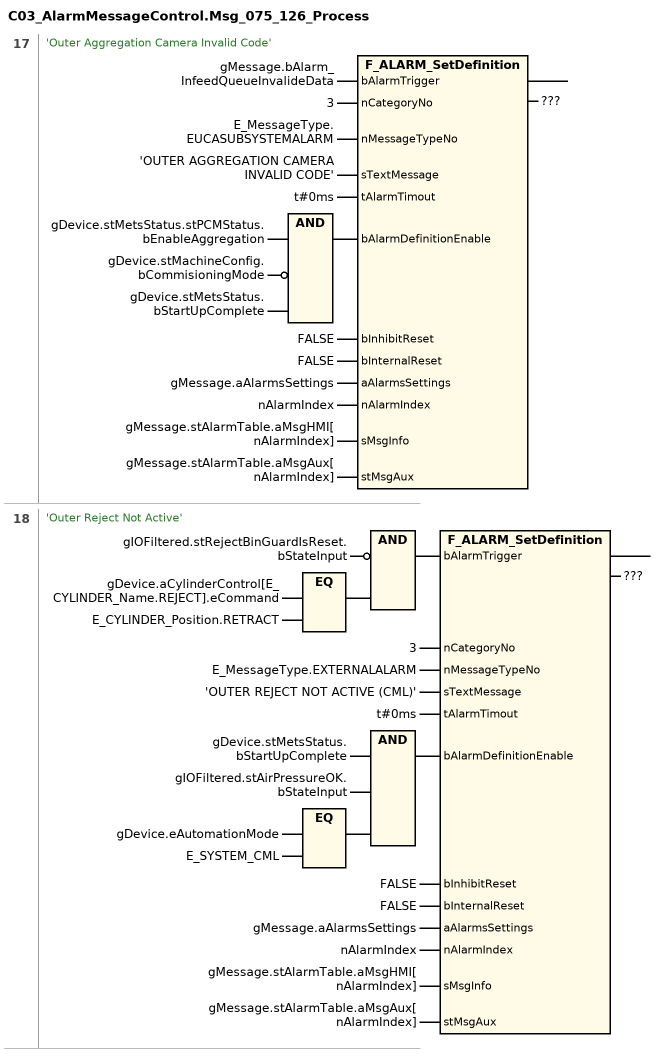
// NETWORK 17
// 'Outer Aggregation Camera Invalid Code'
F_ALARM_SetDefinition(bAlarmTrigger := gMessage.bAlarm_InfeedQueueInvalideData, nCategoryNo := 3, nMessageTypeNo := E_MessageType.EUCASUBSYSTEMALARM, sTextMessage := 'OUTER AGGREGATION CAMERA INVALID CODE', tAlarmTimout := t#0ms, bAlarmDefinitionEnable := gDevice.stMetsStatus.stPCMStatus.bEnableAggregation AND NOT gDevice.stMachineConfig.bCommisioningMode AND gDevice.stMetsStatus.bStartUpComplete, bInhibitReset := FALSE, bInternalReset := FALSE, aAlarmsSettings := gMessage.aAlarmsSettings, nAlarmIndex := nAlarmIndex, sMsgInfo := gMessage.stAlarmTable.aMsgHMI[nAlarmIndex], stMsgAux := gMessage.stAlarmTable.aMsgAux[nAlarmIndex]);

// NETWORK 18
// 'Outer Reject Not Active'
F_ALARM_SetDefinition(bAlarmTrigger := NOT gIOFiltered.stRejectBinGuardIsReset.bStateInput AND gDevice.aCylinderControl[E_CYLINDER_Name.REJECT].eCommand = E_CYLINDER_Position.RETRACT, nCategoryNo := 3, nMessageTypeNo := E_MessageType.EXTERNALALARM, sTextMessage := 'OUTER REJECT NOT ACTIVE (CML)', tAlarmTimout := t#0ms, bAlarmDefinitionEnable := gDevice.stMetsStatus.bStartUpComplete AND gIOFiltered.stAirPressureOK.bStateInput AND gDevice.eAutomationMode = E_SYSTEM_CML, bInhibitReset := FALSE, bInternalReset := FALSE, aAlarmsSettings := gMessage.aAlarmsSettings, nAlarmIndex := nAlarmIndex, sMsgInfo := gMessage.stAlarmTable.aMsgHMI[nAlarmIndex], stMsgAux := gMessage.stAlarmTable.aMsgAux[nAlarmIndex]);

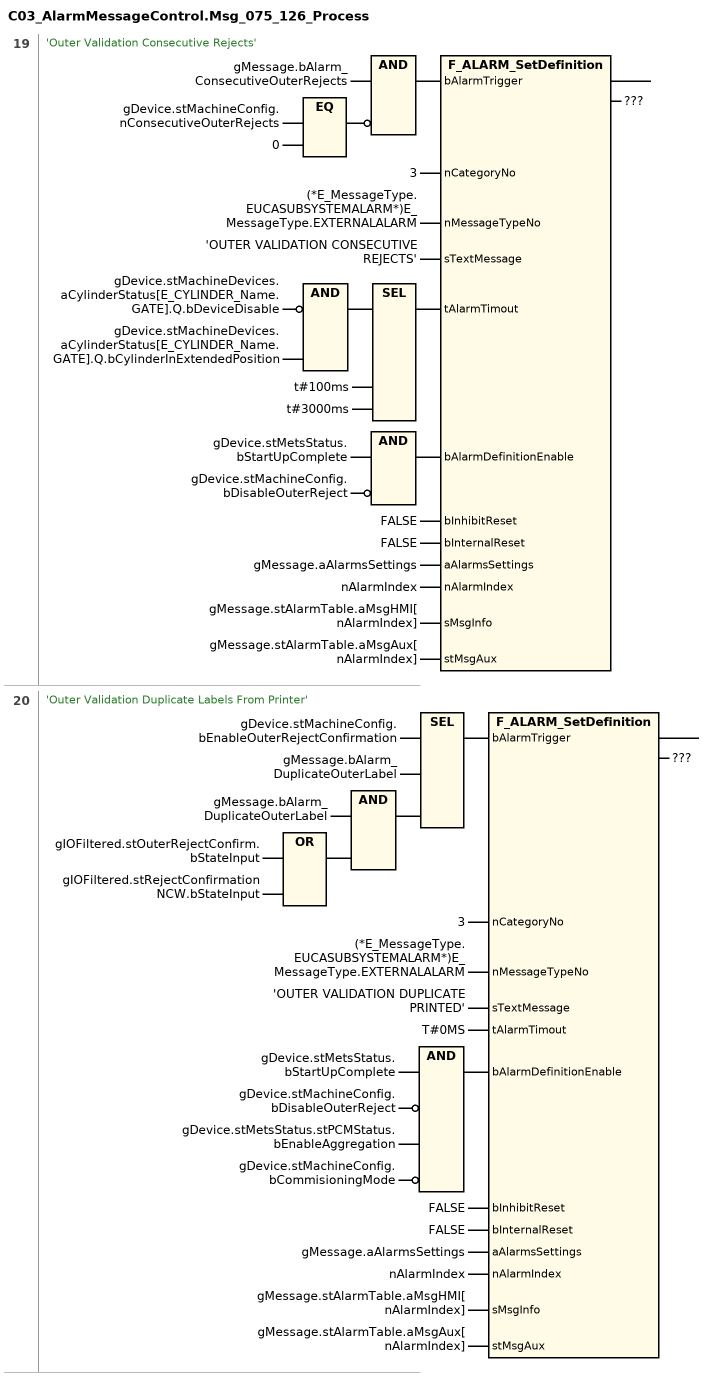
// NETWORK 19
// 'Outer Validation Consecutive Rejects'
F_ALARM_SetDefinition(bAlarmTrigger := gMessage.bAlarm_ConsecutiveOuterRejects AND NOT (gDevice.stMachineConfig.nConsecutiveOuterRejects = 0), nCategoryNo := 3, nMessageTypeNo := (*E_MessageType.EUCASUBSYSTEMALARM*)E_MessageType.EXTERNALALARM, sTextMessage := 'OUTER VALIDATION CONSECUTIVE REJECTS', tAlarmTimout := SEL(NOT gDevice.stMachineDevices.aCylinderStatus[E_CYLINDER_Name.GATE].Q.bDeviceDisable AND gDevice.stMachineDevices.aCylinderStatus[E_CYLINDER_Name.GATE].Q.bCylinderInExtendedPosition, t#100ms, t#3000ms), bAlarmDefinitionEnable := gDevice.stMetsStatus.bStartUpComplete AND NOT gDevice.stMachineConfig.bDisableOuterReject, bInhibitReset := FALSE, bInternalReset := FALSE, aAlarmsSettings := gMessage.aAlarmsSettings, nAlarmIndex := nAlarmIndex, sMsgInfo := gMessage.stAlarmTable.aMsgHMI[nAlarmIndex], stMsgAux := gMessage.stAlarmTable.aMsgAux[nAlarmIndex]);

// NETWORK 20
// 'Outer Validation Duplicate Labels From Printer'
F_ALARM_SetDefinition(bAlarmTrigger := SEL(gDevice.stMachineConfig.bEnableOuterRejectConfirmation, gMessage.bAlarm_DuplicateOuterLabel, gMessage.bAlarm_DuplicateOuterLabel AND (gIOFiltered.stOuterRejectConfirm.bStateInput OR gIOFiltered.stRejectConfirmationNCW.bStateInput)), nCategoryNo := 3, nMessageTypeNo := (*E_MessageType.EUCASUBSYSTEMALARM*)E_MessageType.EXTERNALALARM, sTextMessage := 'OUTER VALIDATION DUPLICATE PRINTED', tAlarmTimout := T#0MS, bAlarmDefinitionEnable := gDevice.stMetsStatus.bStartUpComplete AND NOT gDevice.stMachineConfig.bDisableOuterReject AND gDevice.stMetsStatus.stPCMStatus.bEnableAggregation AND NOT gDevice.stMachineConfig.bCommisioningMode, bInhibitReset := FALSE, bInternalReset := FALSE, aAlarmsSettings := gMessage.aAlarmsSettings, nAlarmIndex := nAlarmIndex, sMsgInfo := gMessage.stAlarmTable.aMsgHMI[nAlarmIndex], stMsgAux := gMessage.stAlarmTable.aMsgAux[nAlarmIndex]);

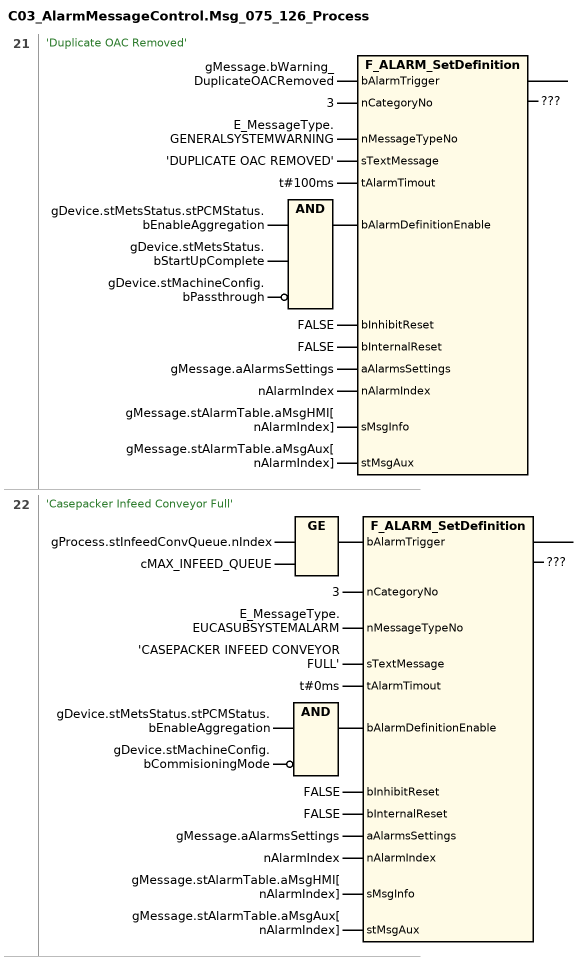
// NETWORK 21
// 'Duplicate OAC Removed'
F_ALARM_SetDefinition(bAlarmTrigger := gMessage.bWarning_DuplicateOACRemoved, nCategoryNo := 3, nMessageTypeNo := E_MessageType.GENERALSYSTEMWARNING, sTextMessage := 'DUPLICATE OAC REMOVED', tAlarmTimout := t#100ms, bAlarmDefinitionEnable := gDevice.stMetsStatus.stPCMStatus.bEnableAggregation AND gDevice.stMetsStatus.bStartUpComplete AND NOT gDevice.stMachineConfig.bPassthrough, bInhibitReset := FALSE, bInternalReset := FALSE, aAlarmsSettings := gMessage.aAlarmsSettings, nAlarmIndex := nAlarmIndex, sMsgInfo := gMessage.stAlarmTable.aMsgHMI[nAlarmIndex], stMsgAux := gMessage.stAlarmTable.aMsgAux[nAlarmIndex]);

// NETWORK 22
// 'Casepacker Infeed Conveyor Full'
F_ALARM_SetDefinition(bAlarmTrigger := gProcess.stInfeedConvQueue.nIndex >= cMAX_INFEED_QUEUE, nCategoryNo := 3, nMessageTypeNo := E_MessageType.EUCASUBSYSTEMALARM, sTextMessage := 'CASEPACKER INFEED CONVEYOR FULL', tAlarmTimout := t#0ms, bAlarmDefinitionEnable := gDevice.stMetsStatus.stPCMStatus.bEnableAggregation AND NOT gDevice.stMachineConfig.bCommisioningMode, bInhibitReset := FALSE, bInternalReset := FALSE, aAlarmsSettings := gMessage.aAlarmsSettings, nAlarmIndex := nAlarmIndex, sMsgInfo := gMessage.stAlarmTable.aMsgHMI[nAlarmIndex], stMsgAux := gMessage.stAlarmTable.aMsgAux[nAlarmIndex]);

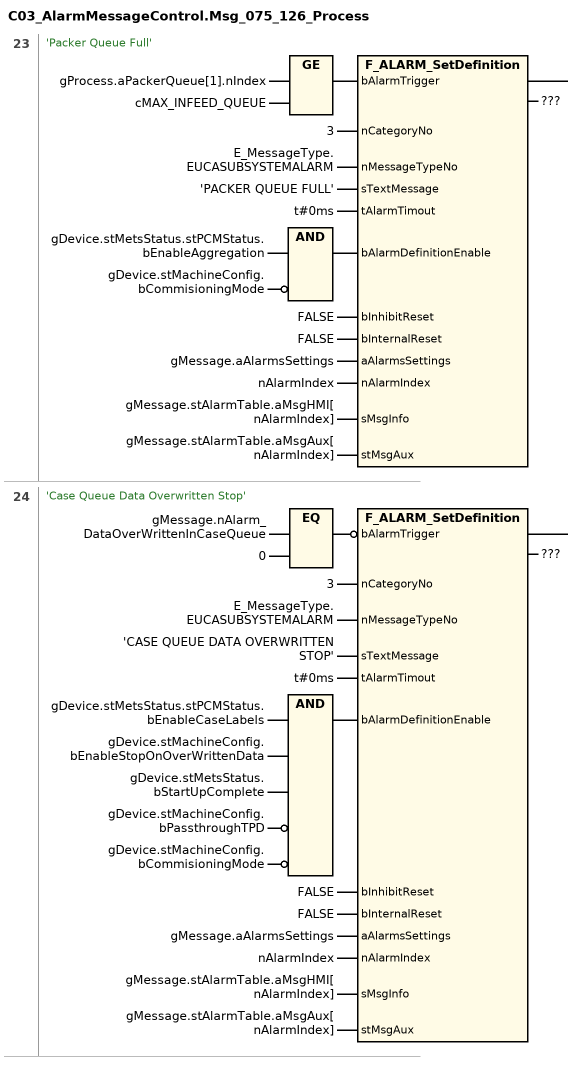
// NETWORK 23
// 'Packer Queue Full'
F_ALARM_SetDefinition(bAlarmTrigger := gProcess.aPackerQueue[1].nIndex >= cMAX_INFEED_QUEUE, nCategoryNo := 3, nMessageTypeNo := E_MessageType.EUCASUBSYSTEMALARM, sTextMessage := 'PACKER QUEUE FULL', tAlarmTimout := t#0ms, bAlarmDefinitionEnable := gDevice.stMetsStatus.stPCMStatus.bEnableAggregation AND NOT gDevice.stMachineConfig.bCommisioningMode, bInhibitReset := FALSE, bInternalReset := FALSE, aAlarmsSettings := gMessage.aAlarmsSettings, nAlarmIndex := nAlarmIndex, sMsgInfo := gMessage.stAlarmTable.aMsgHMI[nAlarmIndex], stMsgAux := gMessage.stAlarmTable.aMsgAux[nAlarmIndex]);

// NETWORK 24
// 'Case Queue Data Overwritten Stop'
F_ALARM_SetDefinition(bAlarmTrigger := NOT (gMessage.nAlarm_DataOverWrittenInCaseQueue = 0), nCategoryNo := 3, nMessageTypeNo := E_MessageType.EUCASUBSYSTEMALARM, sTextMessage := 'CASE QUEUE DATA OVERWRITTEN STOP', tAlarmTimout := t#0ms, bAlarmDefinitionEnable := gDevice.stMetsStatus.stPCMStatus.bEnableCaseLabels AND gDevice.stMachineConfig.bEnableStopOnOverWrittenData AND gDevice.stMetsStatus.bStartUpComplete AND NOT gDevice.stMachineConfig.bPassthroughTPD AND NOT gDevice.stMachineConfig.bCommisioningMode, bInhibitReset := FALSE, bInternalReset := FALSE, aAlarmsSettings := gMessage.aAlarmsSettings, nAlarmIndex := nAlarmIndex, sMsgInfo := gMessage.stAlarmTable.aMsgHMI[nAlarmIndex], stMsgAux := gMessage.stAlarmTable.aMsgAux[nAlarmIndex]);

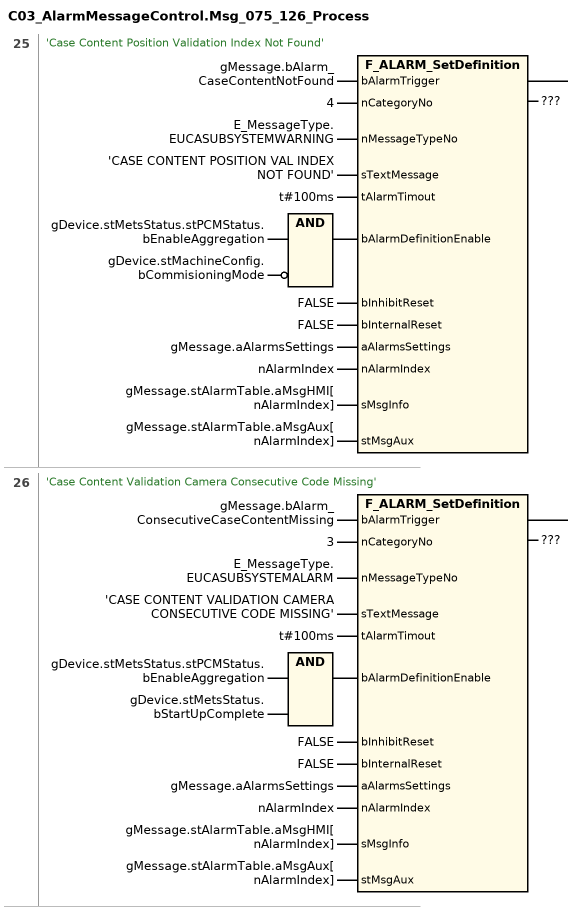
// NETWORK 25
// 'Case Content Position Validation Index Not Found'
F_ALARM_SetDefinition(bAlarmTrigger := gMessage.bAlarm_CaseContentNotFound, nCategoryNo := 4, nMessageTypeNo := E_MessageType.EUCASUBSYSTEMWARNING, sTextMessage := 'CASE CONTENT POSITION VAL INDEX NOT FOUND', tAlarmTimout := t#100ms, bAlarmDefinitionEnable := gDevice.stMetsStatus.stPCMStatus.bEnableAggregation AND NOT gDevice.stMachineConfig.bCommisioningMode, bInhibitReset := FALSE, bInternalReset := FALSE, aAlarmsSettings := gMessage.aAlarmsSettings, nAlarmIndex := nAlarmIndex, sMsgInfo := gMessage.stAlarmTable.aMsgHMI[nAlarmIndex], stMsgAux := gMessage.stAlarmTable.aMsgAux[nAlarmIndex]);

// NETWORK 26
// 'Case Content Validation Camera Consecutive Code Missing'
F_ALARM_SetDefinition(bAlarmTrigger := gMessage.bAlarm_ConsecutiveCaseContentMissing, nCategoryNo := 3, nMessageTypeNo := E_MessageType.EUCASUBSYSTEMALARM, sTextMessage := 'CASE CONTENT VALIDATION CAMERA CONSECUTIVE CODE MISSING', tAlarmTimout := t#100ms, bAlarmDefinitionEnable := gDevice.stMetsStatus.stPCMStatus.bEnableAggregation AND gDevice.stMetsStatus.bStartUpComplete, bInhibitReset := FALSE, bInternalReset := FALSE, aAlarmsSettings := gMessage.aAlarmsSettings, nAlarmIndex := nAlarmIndex, sMsgInfo := gMessage.stAlarmTable.aMsgHMI[nAlarmIndex], stMsgAux := gMessage.stAlarmTable.aMsgAux[nAlarmIndex]);

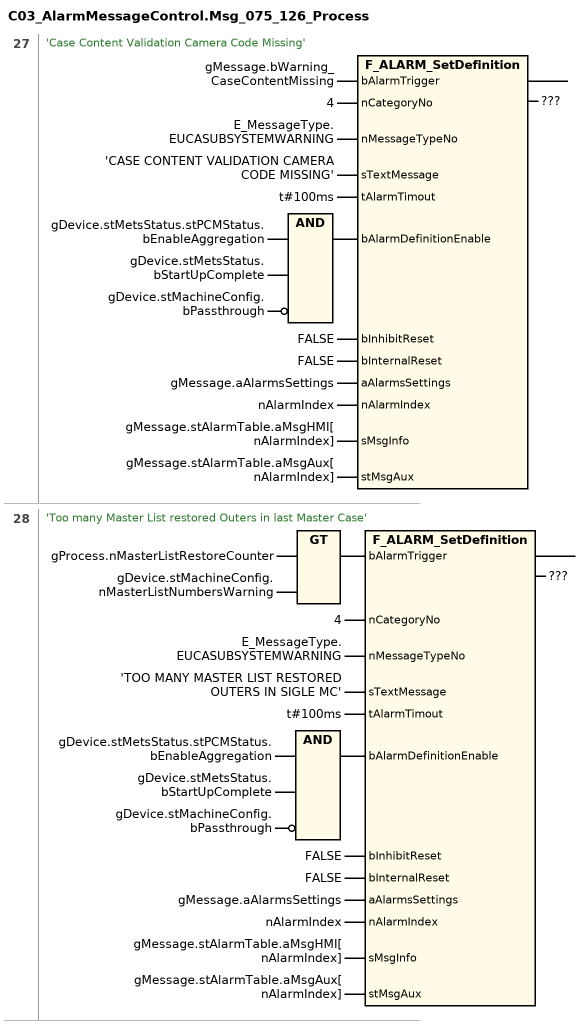
// NETWORK 27
// 'Case Content Validation Camera Code Missing'
F_ALARM_SetDefinition(bAlarmTrigger := gMessage.bWarning_CaseContentMissing, nCategoryNo := 4, nMessageTypeNo := E_MessageType.EUCASUBSYSTEMWARNING, sTextMessage := 'CASE CONTENT VALIDATION CAMERA CODE MISSING', tAlarmTimout := t#100ms, bAlarmDefinitionEnable := gDevice.stMetsStatus.stPCMStatus.bEnableAggregation AND gDevice.stMetsStatus.bStartUpComplete AND NOT gDevice.stMachineConfig.bPassthrough, bInhibitReset := FALSE, bInternalReset := FALSE, aAlarmsSettings := gMessage.aAlarmsSettings, nAlarmIndex := nAlarmIndex, sMsgInfo := gMessage.stAlarmTable.aMsgHMI[nAlarmIndex], stMsgAux := gMessage.stAlarmTable.aMsgAux[nAlarmIndex]);

// NETWORK 28
// 'Too many Master List restored Outers in last Master Case'
F_ALARM_SetDefinition(bAlarmTrigger := gProcess.nMasterListRestoreCounter > gDevice.stMachineConfig.nMasterListNumbersWarning, nCategoryNo := 4, nMessageTypeNo := E_MessageType.EUCASUBSYSTEMWARNING, sTextMessage := 'TOO MANY MASTER LIST RESTORED OUTERS IN SIGLE MC', tAlarmTimout := t#100ms, bAlarmDefinitionEnable := gDevice.stMetsStatus.stPCMStatus.bEnableAggregation AND gDevice.stMetsStatus.bStartUpComplete AND NOT gDevice.stMachineConfig.bPassthrough, bInhibitReset := FALSE, bInternalReset := FALSE, aAlarmsSettings := gMessage.aAlarmsSettings, nAlarmIndex := nAlarmIndex, sMsgInfo := gMessage.stAlarmTable.aMsgHMI[nAlarmIndex], stMsgAux := gMessage.stAlarmTable.aMsgAux[nAlarmIndex]);

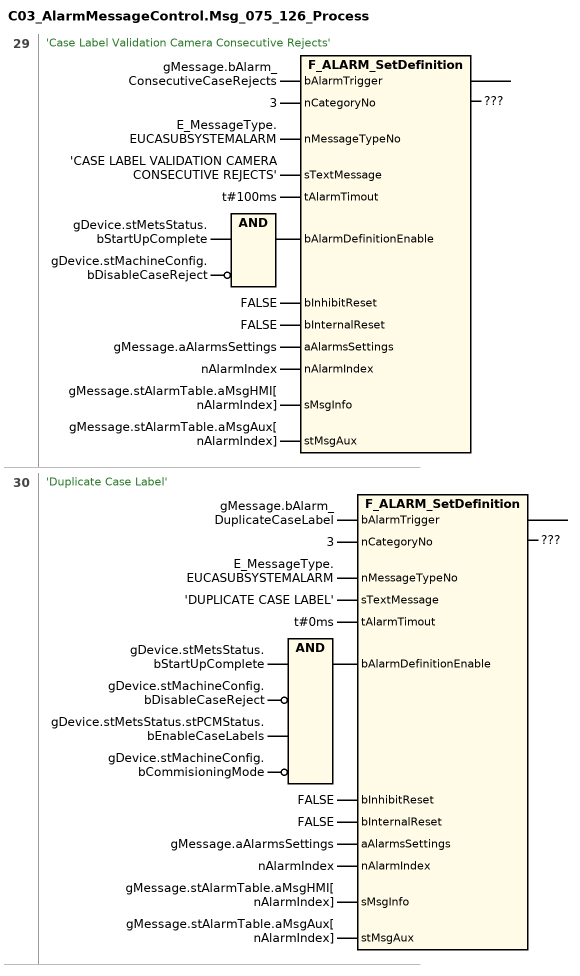
// NETWORK 29
// 'Case Label Validation Camera Consecutive Rejects'
F_ALARM_SetDefinition(bAlarmTrigger := gMessage.bAlarm_ConsecutiveCaseRejects, nCategoryNo := 3, nMessageTypeNo := E_MessageType.EUCASUBSYSTEMALARM, sTextMessage := 'CASE LABEL VALIDATION CAMERA CONSECUTIVE REJECTS', tAlarmTimout := t#100ms, bAlarmDefinitionEnable := gDevice.stMetsStatus.bStartUpComplete AND NOT gDevice.stMachineConfig.bDisableCaseReject, bInhibitReset := FALSE, bInternalReset := FALSE, aAlarmsSettings := gMessage.aAlarmsSettings, nAlarmIndex := nAlarmIndex, sMsgInfo := gMessage.stAlarmTable.aMsgHMI[nAlarmIndex], stMsgAux := gMessage.stAlarmTable.aMsgAux[nAlarmIndex]);

// NETWORK 30
// 'Duplicate Case Label'
F_ALARM_SetDefinition(bAlarmTrigger := gMessage.bAlarm_DuplicateCaseLabel, nCategoryNo := 3, nMessageTypeNo := E_MessageType.EUCASUBSYSTEMALARM, sTextMessage := 'DUPLICATE CASE LABEL', tAlarmTimout := t#0ms, bAlarmDefinitionEnable := gDevice.stMetsStatus.bStartUpComplete AND NOT gDevice.stMachineConfig.bDisableCaseReject AND gDevice.stMetsStatus.stPCMStatus.bEnableCaseLabels AND NOT gDevice.stMachineConfig.bCommisioningMode, bInhibitReset := FALSE, bInternalReset := FALSE, aAlarmsSettings := gMessage.aAlarmsSettings, nAlarmIndex := nAlarmIndex, sMsgInfo := gMessage.stAlarmTable.aMsgHMI[nAlarmIndex], stMsgAux := gMessage.stAlarmTable.aMsgAux[nAlarmIndex]);

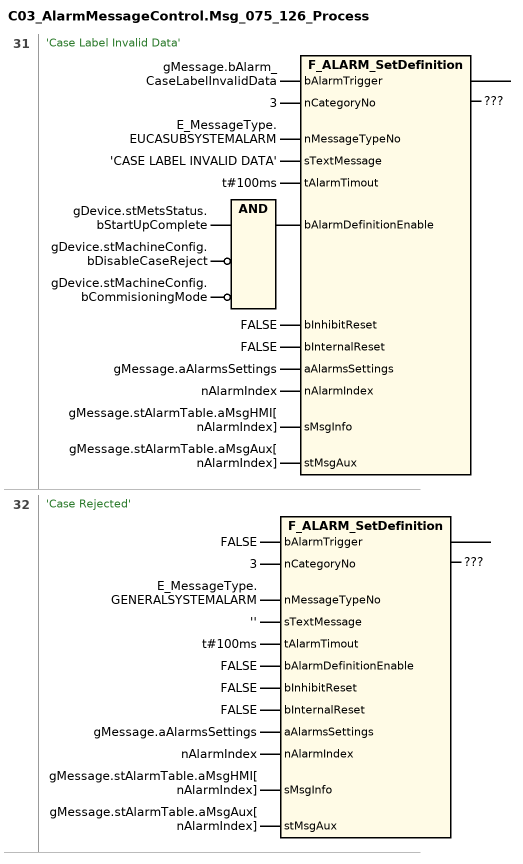
// NETWORK 31
// 'Case Label Invalid Data'
F_ALARM_SetDefinition(bAlarmTrigger := gMessage.bAlarm_CaseLabelInvalidData, nCategoryNo := 3, nMessageTypeNo := E_MessageType.EUCASUBSYSTEMALARM, sTextMessage := 'CASE LABEL INVALID DATA', tAlarmTimout := t#100ms, bAlarmDefinitionEnable := gDevice.stMetsStatus.bStartUpComplete AND NOT gDevice.stMachineConfig.bDisableCaseReject AND NOT gDevice.stMachineConfig.bCommisioningMode, bInhibitReset := FALSE, bInternalReset := FALSE, aAlarmsSettings := gMessage.aAlarmsSettings, nAlarmIndex := nAlarmIndex, sMsgInfo := gMessage.stAlarmTable.aMsgHMI[nAlarmIndex], stMsgAux := gMessage.stAlarmTable.aMsgAux[nAlarmIndex]);

// NETWORK 32
// 'Case Rejected'
F_ALARM_SetDefinition(bAlarmTrigger := FALSE, nCategoryNo := 3, nMessageTypeNo := E_MessageType.GENERALSYSTEMALARM, sTextMessage := '', tAlarmTimout := t#100ms, bAlarmDefinitionEnable := FALSE, bInhibitReset := FALSE, bInternalReset := FALSE, aAlarmsSettings := gMessage.aAlarmsSettings, nAlarmIndex := nAlarmIndex, sMsgInfo := gMessage.stAlarmTable.aMsgHMI[nAlarmIndex], stMsgAux := gMessage.stAlarmTable.aMsgAux[nAlarmIndex]);

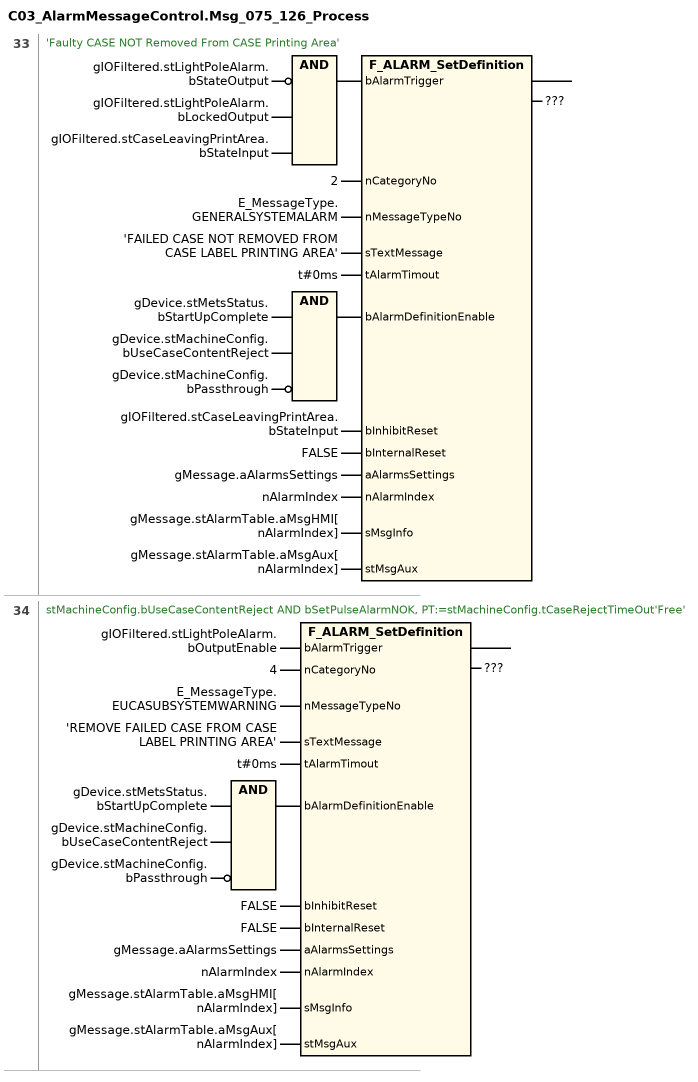
// NETWORK 33
// 'Faulty CASE NOT Removed From CASE Printing Area'
F_ALARM_SetDefinition(bAlarmTrigger := NOT gIOFiltered.stLightPoleAlarm.bStateOutput AND gIOFiltered.stLightPoleAlarm.bLockedOutput AND gIOFiltered.stCaseLeavingPrintArea.bStateInput, nCategoryNo := 2, nMessageTypeNo := E_MessageType.GENERALSYSTEMALARM, sTextMessage := 'FAILED CASE NOT REMOVED FROM CASE LABEL PRINTING AREA', tAlarmTimout := t#0ms, bAlarmDefinitionEnable := gDevice.stMetsStatus.bStartUpComplete AND gDevice.stMachineConfig.bUseCaseContentReject AND NOT gDevice.stMachineConfig.bPassthrough, bInhibitReset := gIOFiltered.stCaseLeavingPrintArea.bStateInput, bInternalReset := FALSE, aAlarmsSettings := gMessage.aAlarmsSettings, nAlarmIndex := nAlarmIndex, sMsgInfo := gMessage.stAlarmTable.aMsgHMI[nAlarmIndex], stMsgAux := gMessage.stAlarmTable.aMsgAux[nAlarmIndex]);

// NETWORK 34
// stMachineConfig.bUseCaseContentReject AND bSetPulseAlarmNOK, PT:=stMachineConfig.tCaseRejectTimeOut'Free'
F_ALARM_SetDefinition(bAlarmTrigger := gIOFiltered.stLightPoleAlarm.bOutputEnable, nCategoryNo := 4, nMessageTypeNo := E_MessageType.EUCASUBSYSTEMWARNING, sTextMessage := 'REMOVE FAILED CASE FROM CASE LABEL PRINTING AREA', tAlarmTimout := t#0ms, bAlarmDefinitionEnable := gDevice.stMetsStatus.bStartUpComplete AND gDevice.stMachineConfig.bUseCaseContentReject AND NOT gDevice.stMachineConfig.bPassthrough, bInhibitReset := FALSE, bInternalReset := FALSE, aAlarmsSettings := gMessage.aAlarmsSettings, nAlarmIndex := nAlarmIndex, sMsgInfo := gMessage.stAlarmTable.aMsgHMI[nAlarmIndex], stMsgAux := gMessage.stAlarmTable.aMsgAux[nAlarmIndex]);

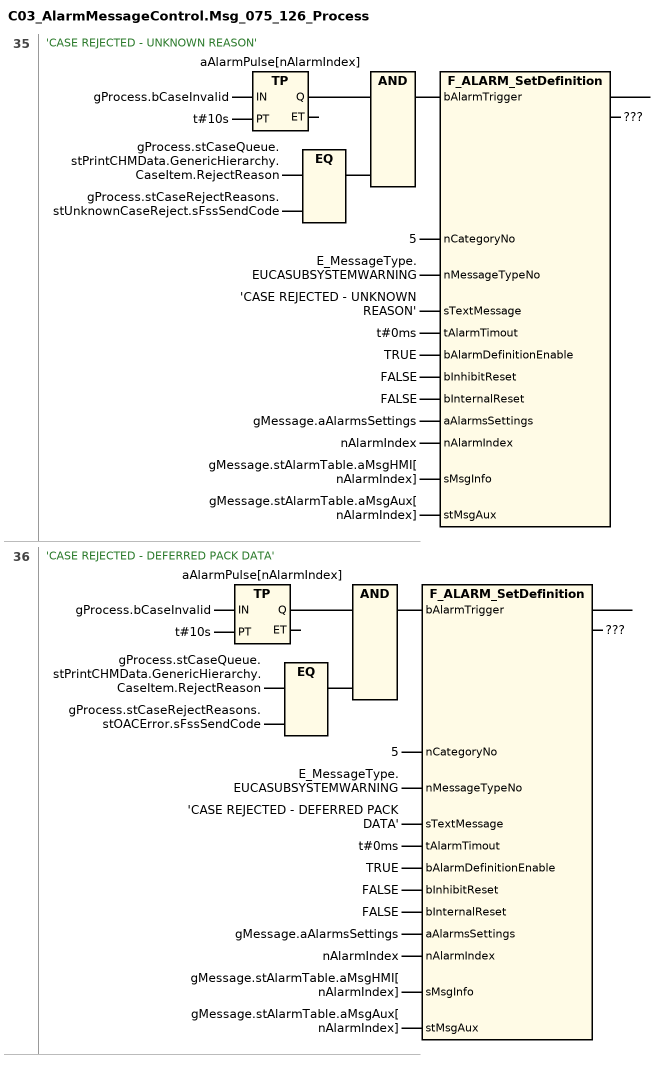
// NETWORK 35
// 'CASE REJECTED - UNKNOWN REASON'
aAlarmPulse[nAlarmIndex](IN := gProcess.bCaseInvalid, PT := t#10s); // TP
F_ALARM_SetDefinition(bAlarmTrigger := aAlarmPulse[nAlarmIndex].Q AND gProcess.stCaseQueue.stPrintCHMData.GenericHierarchy.CaseItem.RejectReason = gProcess.stCaseRejectReasons.stUnknownCaseReject.sFssSendCode, nCategoryNo := 5, nMessageTypeNo := E_MessageType.EUCASUBSYSTEMWARNING, sTextMessage := 'CASE REJECTED - UNKNOWN REASON', tAlarmTimout := t#0ms, bAlarmDefinitionEnable := TRUE, bInhibitReset := FALSE, bInternalReset := FALSE, aAlarmsSettings := gMessage.aAlarmsSettings, nAlarmIndex := nAlarmIndex, sMsgInfo := gMessage.stAlarmTable.aMsgHMI[nAlarmIndex], stMsgAux := gMessage.stAlarmTable.aMsgAux[nAlarmIndex]);

// NETWORK 36
// 'CASE REJECTED - DEFERRED PACK DATA'
aAlarmPulse[nAlarmIndex](IN := gProcess.bCaseInvalid, PT := t#10s); // TP
F_ALARM_SetDefinition(bAlarmTrigger := aAlarmPulse[nAlarmIndex].Q AND gProcess.stCaseQueue.stPrintCHMData.GenericHierarchy.CaseItem.RejectReason = gProcess.stCaseRejectReasons.stOACError.sFssSendCode, nCategoryNo := 5, nMessageTypeNo := E_MessageType.EUCASUBSYSTEMWARNING, sTextMessage := 'CASE REJECTED - DEFERRED PACK DATA', tAlarmTimout := t#0ms, bAlarmDefinitionEnable := TRUE, bInhibitReset := FALSE, bInternalReset := FALSE, aAlarmsSettings := gMessage.aAlarmsSettings, nAlarmIndex := nAlarmIndex, sMsgInfo := gMessage.stAlarmTable.aMsgHMI[nAlarmIndex], stMsgAux := gMessage.stAlarmTable.aMsgAux[nAlarmIndex]);

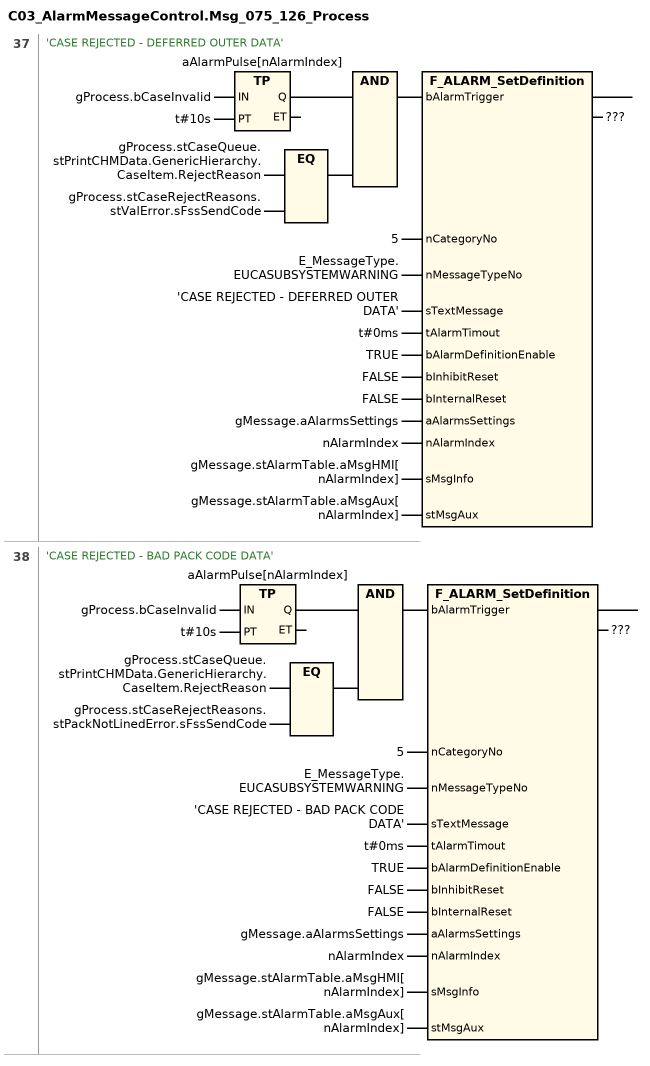
// NETWORK 37
// 'CASE REJECTED - DEFERRED OUTER DATA'
aAlarmPulse[nAlarmIndex](IN := gProcess.bCaseInvalid, PT := t#10s); // TP
F_ALARM_SetDefinition(bAlarmTrigger := aAlarmPulse[nAlarmIndex].Q AND gProcess.stCaseQueue.stPrintCHMData.GenericHierarchy.CaseItem.RejectReason = gProcess.stCaseRejectReasons.stValError.sFssSendCode, nCategoryNo := 5, nMessageTypeNo := E_MessageType.EUCASUBSYSTEMWARNING, sTextMessage := 'CASE REJECTED - DEFERRED OUTER DATA', tAlarmTimout := t#0ms, bAlarmDefinitionEnable := TRUE, bInhibitReset := FALSE, bInternalReset := FALSE, aAlarmsSettings := gMessage.aAlarmsSettings, nAlarmIndex := nAlarmIndex, sMsgInfo := gMessage.stAlarmTable.aMsgHMI[nAlarmIndex], stMsgAux := gMessage.stAlarmTable.aMsgAux[nAlarmIndex]);

// NETWORK 38
// 'CASE REJECTED - BAD PACK CODE DATA'
aAlarmPulse[nAlarmIndex](IN := gProcess.bCaseInvalid, PT := t#10s); // TP
F_ALARM_SetDefinition(bAlarmTrigger := aAlarmPulse[nAlarmIndex].Q AND gProcess.stCaseQueue.stPrintCHMData.GenericHierarchy.CaseItem.RejectReason = gProcess.stCaseRejectReasons.stPackNotLinedError.sFssSendCode, nCategoryNo := 5, nMessageTypeNo := E_MessageType.EUCASUBSYSTEMWARNING, sTextMessage := 'CASE REJECTED - BAD PACK CODE DATA', tAlarmTimout := t#0ms, bAlarmDefinitionEnable := TRUE, bInhibitReset := FALSE, bInternalReset := FALSE, aAlarmsSettings := gMessage.aAlarmsSettings, nAlarmIndex := nAlarmIndex, sMsgInfo := gMessage.stAlarmTable.aMsgHMI[nAlarmIndex], stMsgAux := gMessage.stAlarmTable.aMsgAux[nAlarmIndex]);

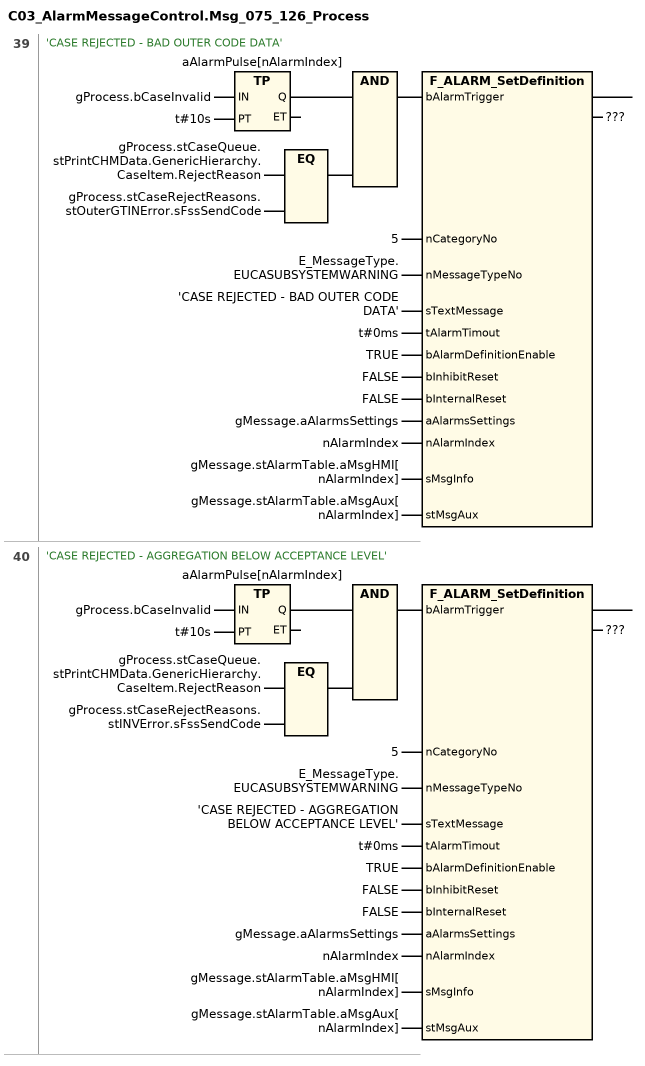
// NETWORK 39
// 'CASE REJECTED - BAD OUTER CODE DATA'
aAlarmPulse[nAlarmIndex](IN := gProcess.bCaseInvalid, PT := t#10s); // TP
F_ALARM_SetDefinition(bAlarmTrigger := aAlarmPulse[nAlarmIndex].Q AND gProcess.stCaseQueue.stPrintCHMData.GenericHierarchy.CaseItem.RejectReason = gProcess.stCaseRejectReasons.stOuterGTINError.sFssSendCode, nCategoryNo := 5, nMessageTypeNo := E_MessageType.EUCASUBSYSTEMWARNING, sTextMessage := 'CASE REJECTED - BAD OUTER CODE DATA', tAlarmTimout := t#0ms, bAlarmDefinitionEnable := TRUE, bInhibitReset := FALSE, bInternalReset := FALSE, aAlarmsSettings := gMessage.aAlarmsSettings, nAlarmIndex := nAlarmIndex, sMsgInfo := gMessage.stAlarmTable.aMsgHMI[nAlarmIndex], stMsgAux := gMessage.stAlarmTable.aMsgAux[nAlarmIndex]);

// NETWORK 40
// 'CASE REJECTED - AGGREGATION BELOW ACCEPTANCE LEVEL'
aAlarmPulse[nAlarmIndex](IN := gProcess.bCaseInvalid, PT := t#10s); // TP
F_ALARM_SetDefinition(bAlarmTrigger := aAlarmPulse[nAlarmIndex].Q AND gProcess.stCaseQueue.stPrintCHMData.GenericHierarchy.CaseItem.RejectReason = gProcess.stCaseRejectReasons.stINVError.sFssSendCode, nCategoryNo := 5, nMessageTypeNo := E_MessageType.EUCASUBSYSTEMWARNING, sTextMessage := 'CASE REJECTED - AGGREGATION BELOW ACCEPTANCE LEVEL', tAlarmTimout := t#0ms, bAlarmDefinitionEnable := TRUE, bInhibitReset := FALSE, bInternalReset := FALSE, aAlarmsSettings := gMessage.aAlarmsSettings, nAlarmIndex := nAlarmIndex, sMsgInfo := gMessage.stAlarmTable.aMsgHMI[nAlarmIndex], stMsgAux := gMessage.stAlarmTable.aMsgAux[nAlarmIndex]);

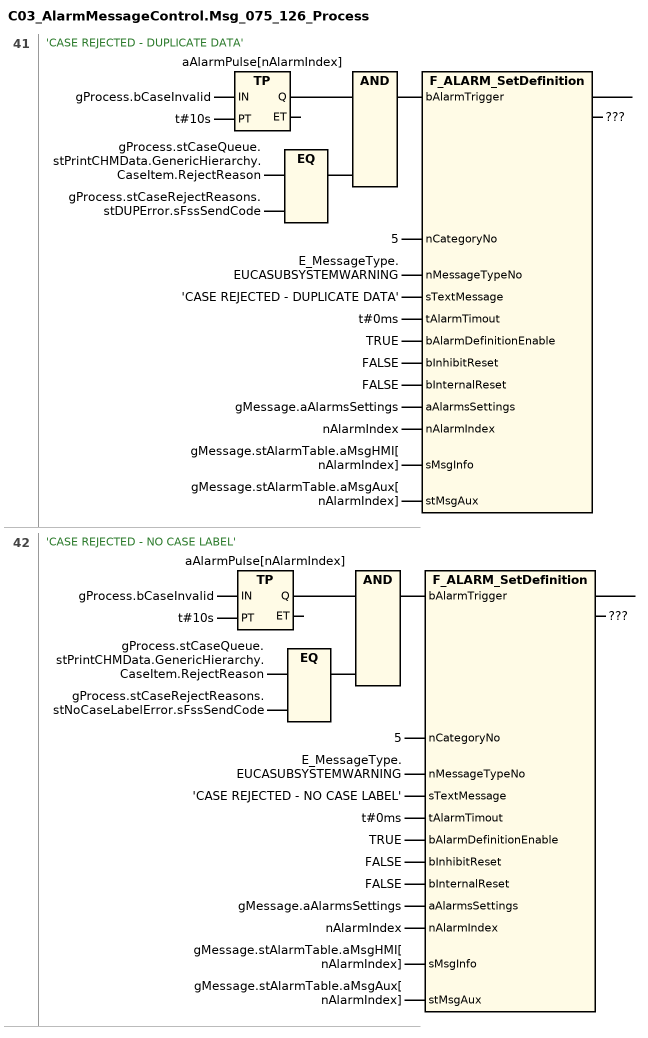
// NETWORK 41
// 'CASE REJECTED - DUPLICATE DATA'
aAlarmPulse[nAlarmIndex](IN := gProcess.bCaseInvalid, PT := t#10s); // TP
F_ALARM_SetDefinition(bAlarmTrigger := aAlarmPulse[nAlarmIndex].Q AND gProcess.stCaseQueue.stPrintCHMData.GenericHierarchy.CaseItem.RejectReason = gProcess.stCaseRejectReasons.stDUPError.sFssSendCode, nCategoryNo := 5, nMessageTypeNo := E_MessageType.EUCASUBSYSTEMWARNING, sTextMessage := 'CASE REJECTED - DUPLICATE DATA', tAlarmTimout := t#0ms, bAlarmDefinitionEnable := TRUE, bInhibitReset := FALSE, bInternalReset := FALSE, aAlarmsSettings := gMessage.aAlarmsSettings, nAlarmIndex := nAlarmIndex, sMsgInfo := gMessage.stAlarmTable.aMsgHMI[nAlarmIndex], stMsgAux := gMessage.stAlarmTable.aMsgAux[nAlarmIndex]);

// NETWORK 42
// 'CASE REJECTED - NO CASE LABEL'
aAlarmPulse[nAlarmIndex](IN := gProcess.bCaseInvalid, PT := t#10s); // TP
F_ALARM_SetDefinition(bAlarmTrigger := aAlarmPulse[nAlarmIndex].Q AND gProcess.stCaseQueue.stPrintCHMData.GenericHierarchy.CaseItem.RejectReason = gProcess.stCaseRejectReasons.stNoCaseLabelError.sFssSendCode, nCategoryNo := 5, nMessageTypeNo := E_MessageType.EUCASUBSYSTEMWARNING, sTextMessage := 'CASE REJECTED - NO CASE LABEL', tAlarmTimout := t#0ms, bAlarmDefinitionEnable := TRUE, bInhibitReset := FALSE, bInternalReset := FALSE, aAlarmsSettings := gMessage.aAlarmsSettings, nAlarmIndex := nAlarmIndex, sMsgInfo := gMessage.stAlarmTable.aMsgHMI[nAlarmIndex], stMsgAux := gMessage.stAlarmTable.aMsgAux[nAlarmIndex]);

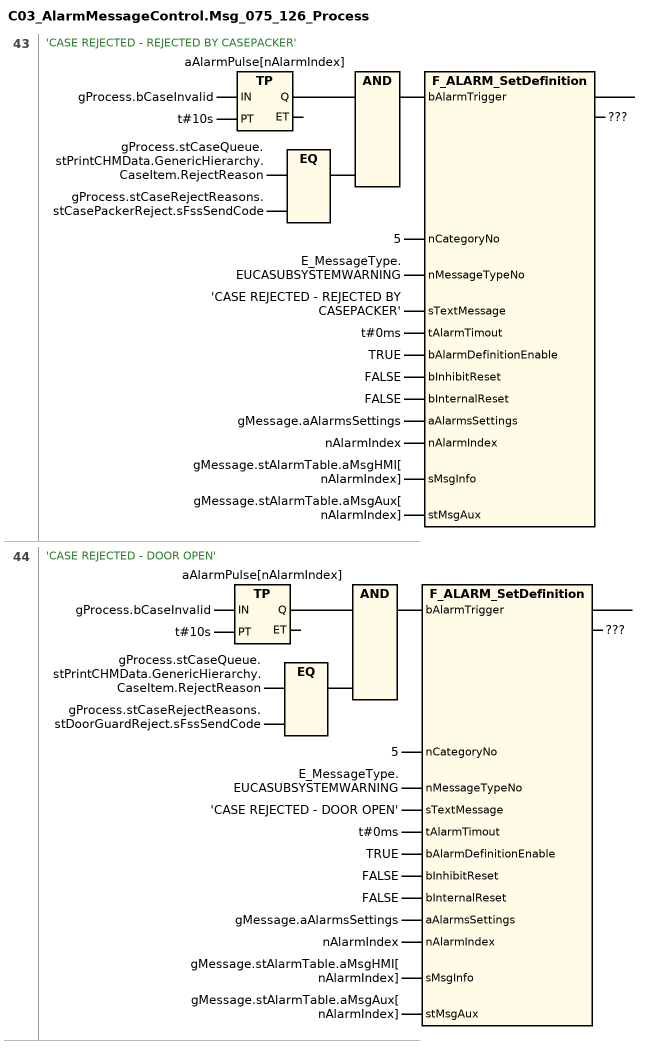
// NETWORK 43
// 'CASE REJECTED - REJECTED BY CASEPACKER'
aAlarmPulse[nAlarmIndex](IN := gProcess.bCaseInvalid, PT := t#10s); // TP
F_ALARM_SetDefinition(bAlarmTrigger := aAlarmPulse[nAlarmIndex].Q AND gProcess.stCaseQueue.stPrintCHMData.GenericHierarchy.CaseItem.RejectReason = gProcess.stCaseRejectReasons.stCasePackerReject.sFssSendCode, nCategoryNo := 5, nMessageTypeNo := E_MessageType.EUCASUBSYSTEMWARNING, sTextMessage := 'CASE REJECTED - REJECTED BY CASEPACKER', tAlarmTimout := t#0ms, bAlarmDefinitionEnable := TRUE, bInhibitReset := FALSE, bInternalReset := FALSE, aAlarmsSettings := gMessage.aAlarmsSettings, nAlarmIndex := nAlarmIndex, sMsgInfo := gMessage.stAlarmTable.aMsgHMI[nAlarmIndex], stMsgAux := gMessage.stAlarmTable.aMsgAux[nAlarmIndex]);

// NETWORK 44
// 'CASE REJECTED - DOOR OPEN'
aAlarmPulse[nAlarmIndex](IN := gProcess.bCaseInvalid, PT := t#10s); // TP
F_ALARM_SetDefinition(bAlarmTrigger := aAlarmPulse[nAlarmIndex].Q AND gProcess.stCaseQueue.stPrintCHMData.GenericHierarchy.CaseItem.RejectReason = gProcess.stCaseRejectReasons.stDoorGuardReject.sFssSendCode, nCategoryNo := 5, nMessageTypeNo := E_MessageType.EUCASUBSYSTEMWARNING, sTextMessage := 'CASE REJECTED - DOOR OPEN', tAlarmTimout := t#0ms, bAlarmDefinitionEnable := TRUE, bInhibitReset := FALSE, bInternalReset := FALSE, aAlarmsSettings := gMessage.aAlarmsSettings, nAlarmIndex := nAlarmIndex, sMsgInfo := gMessage.stAlarmTable.aMsgHMI[nAlarmIndex], stMsgAux := gMessage.stAlarmTable.aMsgAux[nAlarmIndex]);

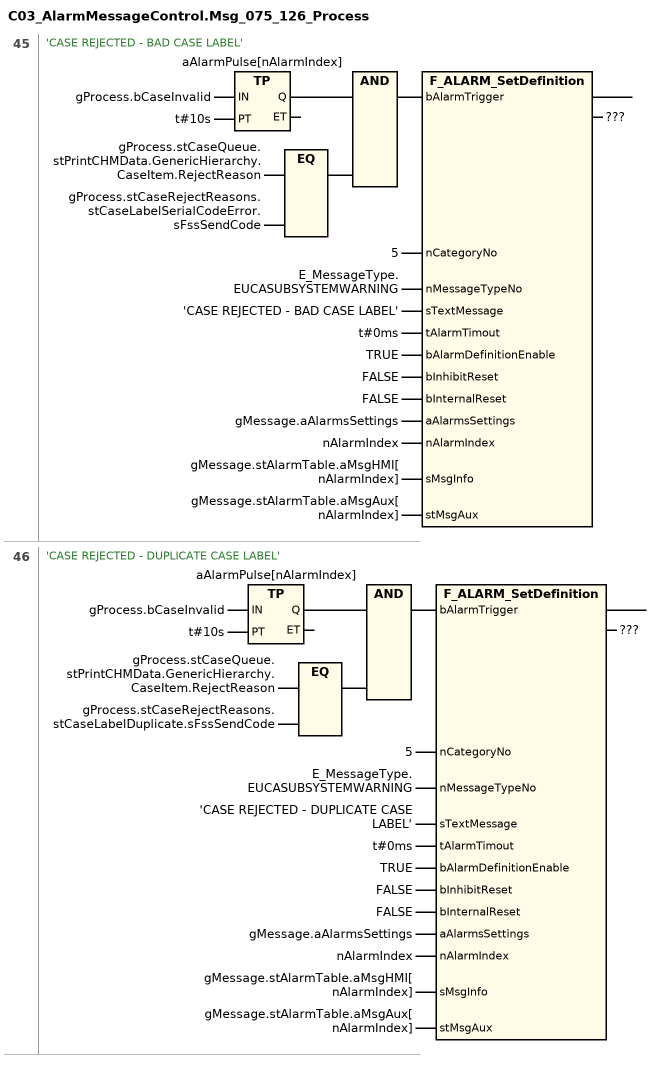
// NETWORK 45
// 'CASE REJECTED - BAD CASE LABEL'
aAlarmPulse[nAlarmIndex](IN := gProcess.bCaseInvalid, PT := t#10s); // TP
F_ALARM_SetDefinition(bAlarmTrigger := aAlarmPulse[nAlarmIndex].Q AND gProcess.stCaseQueue.stPrintCHMData.GenericHierarchy.CaseItem.RejectReason = gProcess.stCaseRejectReasons.stCaseLabelSerialCodeError.sFssSendCode, nCategoryNo := 5, nMessageTypeNo := E_MessageType.EUCASUBSYSTEMWARNING, sTextMessage := 'CASE REJECTED - BAD CASE LABEL', tAlarmTimout := t#0ms, bAlarmDefinitionEnable := TRUE, bInhibitReset := FALSE, bInternalReset := FALSE, aAlarmsSettings := gMessage.aAlarmsSettings, nAlarmIndex := nAlarmIndex, sMsgInfo := gMessage.stAlarmTable.aMsgHMI[nAlarmIndex], stMsgAux := gMessage.stAlarmTable.aMsgAux[nAlarmIndex]);

// NETWORK 46
// 'CASE REJECTED - DUPLICATE CASE LABEL'
aAlarmPulse[nAlarmIndex](IN := gProcess.bCaseInvalid, PT := t#10s); // TP
F_ALARM_SetDefinition(bAlarmTrigger := aAlarmPulse[nAlarmIndex].Q AND gProcess.stCaseQueue.stPrintCHMData.GenericHierarchy.CaseItem.RejectReason = gProcess.stCaseRejectReasons.stCaseLabelDuplicate.sFssSendCode, nCategoryNo := 5, nMessageTypeNo := E_MessageType.EUCASUBSYSTEMWARNING, sTextMessage := 'CASE REJECTED - DUPLICATE CASE LABEL', tAlarmTimout := t#0ms, bAlarmDefinitionEnable := TRUE, bInhibitReset := FALSE, bInternalReset := FALSE, aAlarmsSettings := gMessage.aAlarmsSettings, nAlarmIndex := nAlarmIndex, sMsgInfo := gMessage.stAlarmTable.aMsgHMI[nAlarmIndex], stMsgAux := gMessage.stAlarmTable.aMsgAux[nAlarmIndex]);

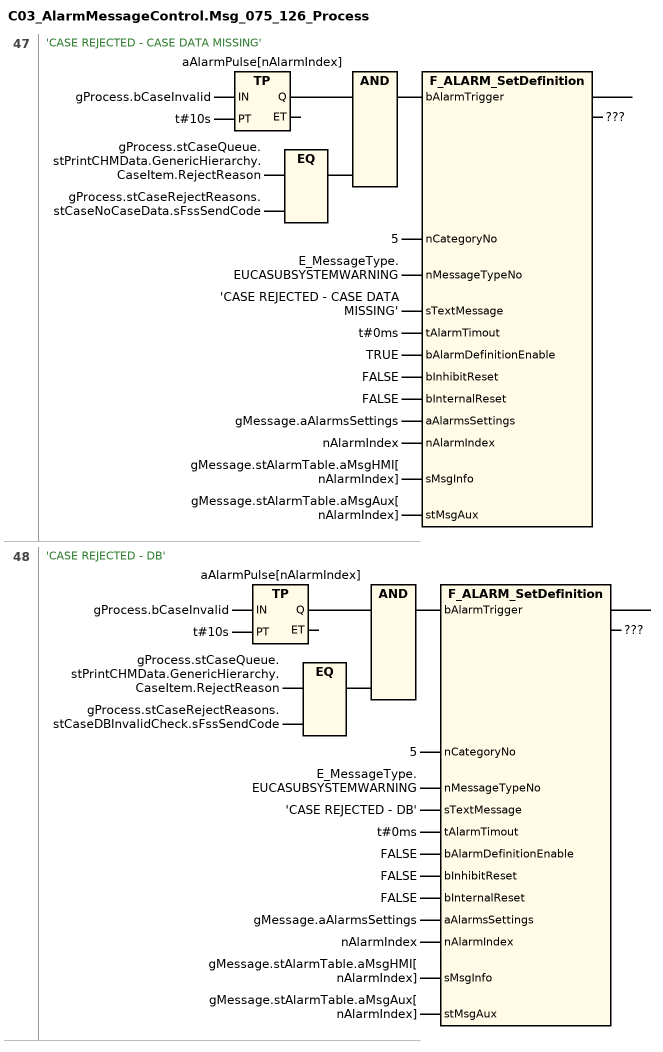
// NETWORK 47
// 'CASE REJECTED - CASE DATA MISSING'
aAlarmPulse[nAlarmIndex](IN := gProcess.bCaseInvalid, PT := t#10s); // TP
F_ALARM_SetDefinition(bAlarmTrigger := aAlarmPulse[nAlarmIndex].Q AND gProcess.stCaseQueue.stPrintCHMData.GenericHierarchy.CaseItem.RejectReason = gProcess.stCaseRejectReasons.stCaseNoCaseData.sFssSendCode, nCategoryNo := 5, nMessageTypeNo := E_MessageType.EUCASUBSYSTEMWARNING, sTextMessage := 'CASE REJECTED - CASE DATA MISSING', tAlarmTimout := t#0ms, bAlarmDefinitionEnable := TRUE, bInhibitReset := FALSE, bInternalReset := FALSE, aAlarmsSettings := gMessage.aAlarmsSettings, nAlarmIndex := nAlarmIndex, sMsgInfo := gMessage.stAlarmTable.aMsgHMI[nAlarmIndex], stMsgAux := gMessage.stAlarmTable.aMsgAux[nAlarmIndex]);

// NETWORK 48
// 'CASE REJECTED - DB'
aAlarmPulse[nAlarmIndex](IN := gProcess.bCaseInvalid, PT := t#10s); // TP
F_ALARM_SetDefinition(bAlarmTrigger := aAlarmPulse[nAlarmIndex].Q AND gProcess.stCaseQueue.stPrintCHMData.GenericHierarchy.CaseItem.RejectReason = gProcess.stCaseRejectReasons.stCaseDBInvalidCheck.sFssSendCode, nCategoryNo := 5, nMessageTypeNo := E_MessageType.EUCASUBSYSTEMWARNING, sTextMessage := 'CASE REJECTED - DB', tAlarmTimout := t#0ms, bAlarmDefinitionEnable := FALSE, bInhibitReset := FALSE, bInternalReset := FALSE, aAlarmsSettings := gMessage.aAlarmsSettings, nAlarmIndex := nAlarmIndex, sMsgInfo := gMessage.stAlarmTable.aMsgHMI[nAlarmIndex], stMsgAux := gMessage.stAlarmTable.aMsgAux[nAlarmIndex]);

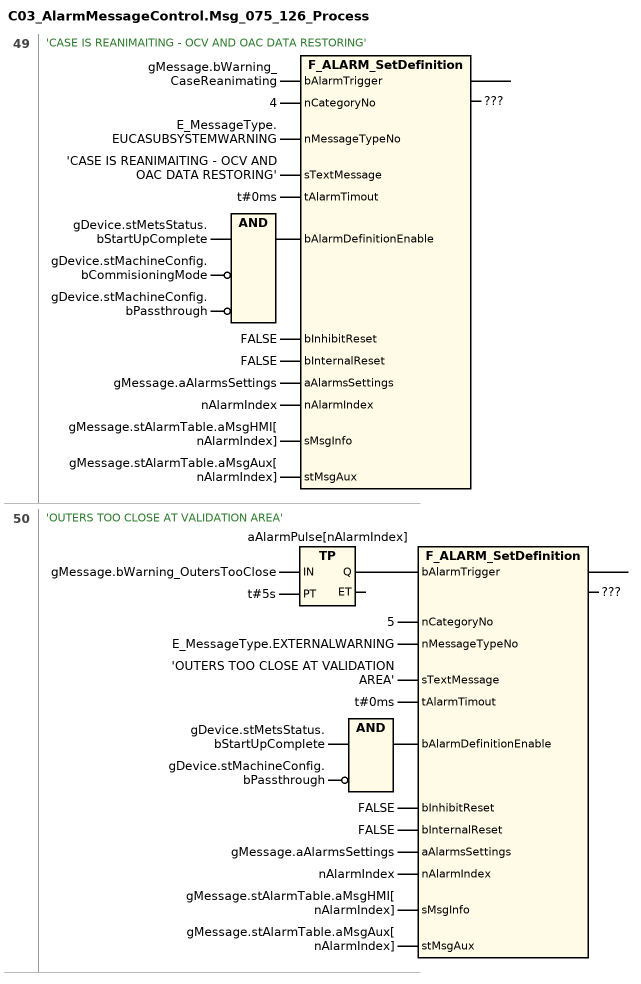
// NETWORK 49
// 'CASE IS REANIMAITING - OCV AND OAC DATA RESTORING'
F_ALARM_SetDefinition(bAlarmTrigger := gMessage.bWarning_CaseReanimating, nCategoryNo := 4, nMessageTypeNo := E_MessageType.EUCASUBSYSTEMWARNING, sTextMessage := 'CASE IS REANIMAITING - OCV AND OAC DATA RESTORING', tAlarmTimout := t#0ms, bAlarmDefinitionEnable := gDevice.stMetsStatus.bStartUpComplete AND NOT gDevice.stMachineConfig.bCommisioningMode AND NOT gDevice.stMachineConfig.bPassthrough, bInhibitReset := FALSE, bInternalReset := FALSE, aAlarmsSettings := gMessage.aAlarmsSettings, nAlarmIndex := nAlarmIndex, sMsgInfo := gMessage.stAlarmTable.aMsgHMI[nAlarmIndex], stMsgAux := gMessage.stAlarmTable.aMsgAux[nAlarmIndex]);

// NETWORK 50
// 'OUTERS TOO CLOSE AT VALIDATION AREA'
aAlarmPulse[nAlarmIndex](IN := gMessage.bWarning_OutersTooClose, PT := t#5s); // TP
F_ALARM_SetDefinition(bAlarmTrigger := aAlarmPulse[nAlarmIndex].Q, nCategoryNo := 5, nMessageTypeNo := E_MessageType.EXTERNALWARNING, sTextMessage := 'OUTERS TOO CLOSE AT VALIDATION AREA', tAlarmTimout := t#0ms, bAlarmDefinitionEnable := gDevice.stMetsStatus.bStartUpComplete AND NOT gDevice.stMachineConfig.bPassthrough, bInhibitReset := FALSE, bInternalReset := FALSE, aAlarmsSettings := gMessage.aAlarmsSettings, nAlarmIndex := nAlarmIndex, sMsgInfo := gMessage.stAlarmTable.aMsgHMI[nAlarmIndex], stMsgAux := gMessage.stAlarmTable.aMsgAux[nAlarmIndex]);

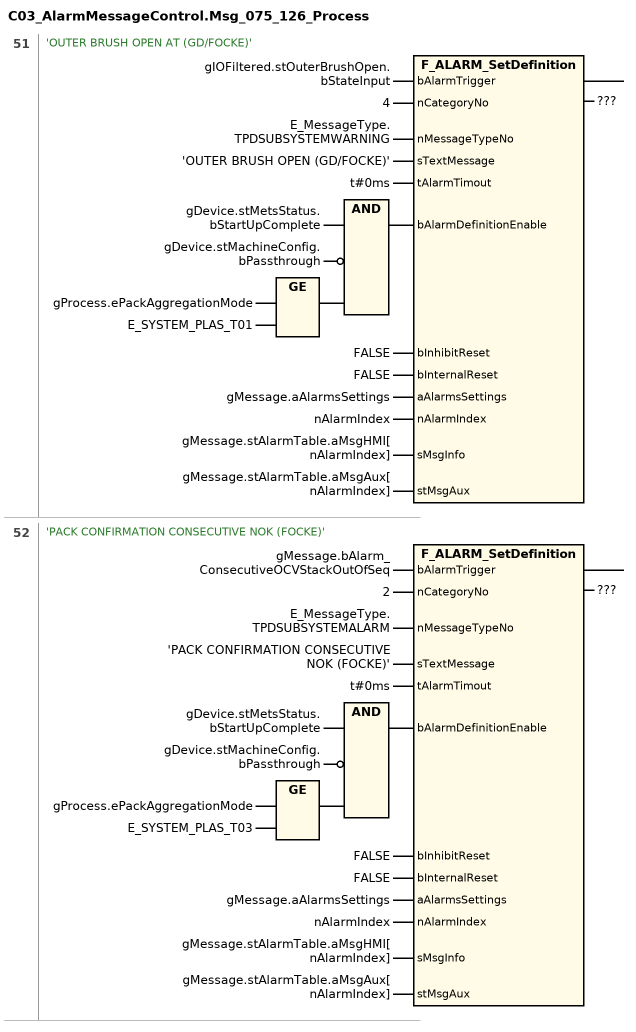
// NETWORK 51
// 'OUTER BRUSH OPEN AT (GD/FOCKE)'
F_ALARM_SetDefinition(bAlarmTrigger := gIOFiltered.stOuterBrushOpen.bStateInput, nCategoryNo := 4, nMessageTypeNo := E_MessageType.TPDSUBSYSTEMWARNING, sTextMessage := 'OUTER BRUSH OPEN (GD/FOCKE)', tAlarmTimout := t#0ms, bAlarmDefinitionEnable := gDevice.stMetsStatus.bStartUpComplete AND NOT gDevice.stMachineConfig.bPassthrough AND gProcess.ePackAggregationMode >= E_SYSTEM_PLAS_T01, bInhibitReset := FALSE, bInternalReset := FALSE, aAlarmsSettings := gMessage.aAlarmsSettings, nAlarmIndex := nAlarmIndex, sMsgInfo := gMessage.stAlarmTable.aMsgHMI[nAlarmIndex], stMsgAux := gMessage.stAlarmTable.aMsgAux[nAlarmIndex]);

// NETWORK 52
// 'PACK CONFIRMATION CONSECUTIVE NOK (FOCKE)'
F_ALARM_SetDefinition(bAlarmTrigger := gMessage.bAlarm_ConsecutiveOCVStackOutOfSeq, nCategoryNo := 2, nMessageTypeNo := E_MessageType.TPDSUBSYSTEMALARM, sTextMessage := 'PACK CONFIRMATION CONSECUTIVE NOK (FOCKE)', tAlarmTimout := t#0ms, bAlarmDefinitionEnable := gDevice.stMetsStatus.bStartUpComplete AND NOT gDevice.stMachineConfig.bPassthrough AND gProcess.ePackAggregationMode >= E_SYSTEM_PLAS_T03, bInhibitReset := FALSE, bInternalReset := FALSE, aAlarmsSettings := gMessage.aAlarmsSettings, nAlarmIndex := nAlarmIndex, sMsgInfo := gMessage.stAlarmTable.aMsgHMI[nAlarmIndex], stMsgAux := gMessage.stAlarmTable.aMsgAux[nAlarmIndex]);
END_ACTION

ACTION Msg_127_150_Sensors:
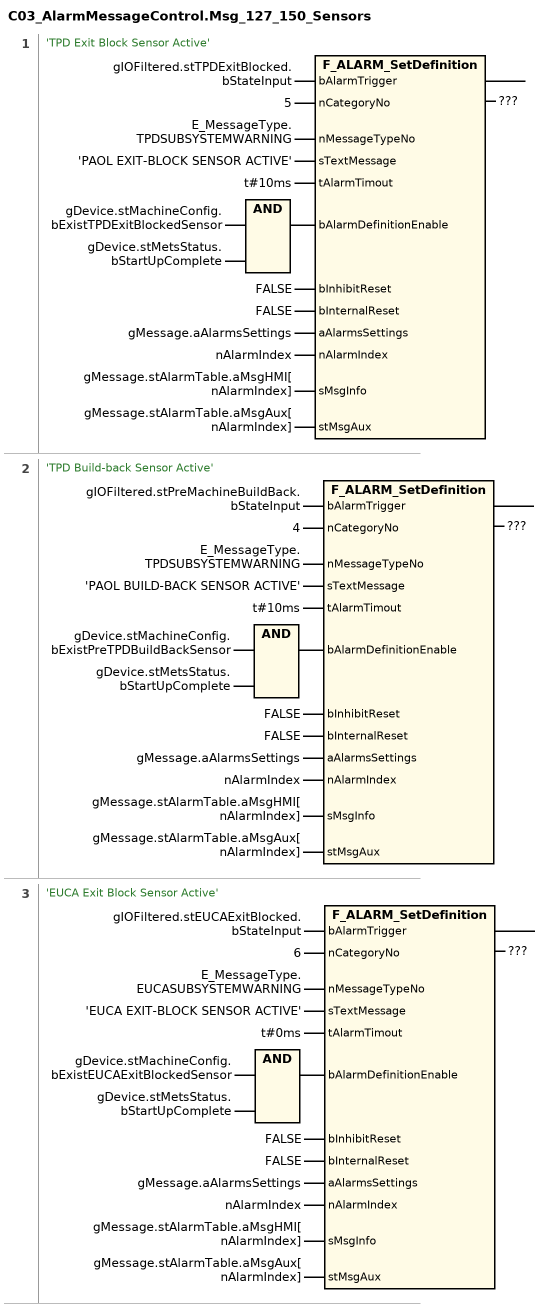
// NETWORK 1
// 'TPD Exit Block Sensor Active'
F_ALARM_SetDefinition(bAlarmTrigger := gIOFiltered.stTPDExitBlocked.bStateInput, nCategoryNo := 5, nMessageTypeNo := E_MessageType.TPDSUBSYSTEMWARNING, sTextMessage := 'PAOL EXIT-BLOCK SENSOR ACTIVE', tAlarmTimout := t#10ms, bAlarmDefinitionEnable := gDevice.stMachineConfig.bExistTPDExitBlockedSensor AND gDevice.stMetsStatus.bStartUpComplete, bInhibitReset := FALSE, bInternalReset := FALSE, aAlarmsSettings := gMessage.aAlarmsSettings, nAlarmIndex := nAlarmIndex, sMsgInfo := gMessage.stAlarmTable.aMsgHMI[nAlarmIndex], stMsgAux := gMessage.stAlarmTable.aMsgAux[nAlarmIndex]);

// NETWORK 2
// 'TPD Build-back Sensor Active'
F_ALARM_SetDefinition(bAlarmTrigger := gIOFiltered.stPreMachineBuildBack.bStateInput, nCategoryNo := 4, nMessageTypeNo := E_MessageType.TPDSUBSYSTEMWARNING, sTextMessage := 'PAOL BUILD-BACK SENSOR ACTIVE', tAlarmTimout := t#10ms, bAlarmDefinitionEnable := gDevice.stMachineConfig.bExistPreTPDBuildBackSensor AND gDevice.stMetsStatus.bStartUpComplete, bInhibitReset := FALSE, bInternalReset := FALSE, aAlarmsSettings := gMessage.aAlarmsSettings, nAlarmIndex := nAlarmIndex, sMsgInfo := gMessage.stAlarmTable.aMsgHMI[nAlarmIndex], stMsgAux := gMessage.stAlarmTable.aMsgAux[nAlarmIndex]);

// NETWORK 3
// 'EUCA Exit Block Sensor Active'
F_ALARM_SetDefinition(bAlarmTrigger := gIOFiltered.stEUCAExitBlocked.bStateInput, nCategoryNo := 6, nMessageTypeNo := E_MessageType.EUCASUBSYSTEMWARNING, sTextMessage := 'EUCA EXIT-BLOCK SENSOR ACTIVE', tAlarmTimout := t#0ms, bAlarmDefinitionEnable := gDevice.stMachineConfig.bExistEUCAExitBlockedSensor AND gDevice.stMetsStatus.bStartUpComplete, bInhibitReset := FALSE, bInternalReset := FALSE, aAlarmsSettings := gMessage.aAlarmsSettings, nAlarmIndex := nAlarmIndex, sMsgInfo := gMessage.stAlarmTable.aMsgHMI[nAlarmIndex], stMsgAux := gMessage.stAlarmTable.aMsgAux[nAlarmIndex]);

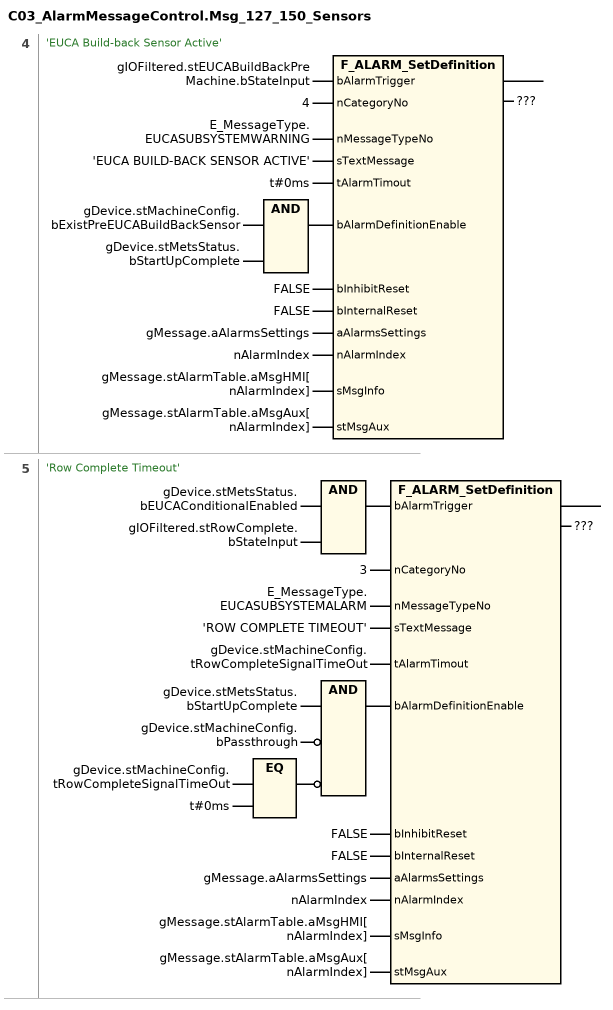
// NETWORK 4
// 'EUCA Build-back Sensor Active'
F_ALARM_SetDefinition(bAlarmTrigger := gIOFiltered.stEUCABuildBackPreMachine.bStateInput, nCategoryNo := 4, nMessageTypeNo := E_MessageType.EUCASUBSYSTEMWARNING, sTextMessage := 'EUCA BUILD-BACK SENSOR ACTIVE', tAlarmTimout := t#0ms, bAlarmDefinitionEnable := gDevice.stMachineConfig.bExistPreEUCABuildBackSensor AND gDevice.stMetsStatus.bStartUpComplete, bInhibitReset := FALSE, bInternalReset := FALSE, aAlarmsSettings := gMessage.aAlarmsSettings, nAlarmIndex := nAlarmIndex, sMsgInfo := gMessage.stAlarmTable.aMsgHMI[nAlarmIndex], stMsgAux := gMessage.stAlarmTable.aMsgAux[nAlarmIndex]);

// NETWORK 5
// 'Row Complete Timeout'
F_ALARM_SetDefinition(bAlarmTrigger := gDevice.stMetsStatus.bEUCAConditionalEnabled AND gIOFiltered.stRowComplete.bStateInput, nCategoryNo := 3, nMessageTypeNo := E_MessageType.EUCASUBSYSTEMALARM, sTextMessage := 'ROW COMPLETE TIMEOUT', tAlarmTimout := gDevice.stMachineConfig.tRowCompleteSignalTimeOut, bAlarmDefinitionEnable := gDevice.stMetsStatus.bStartUpComplete AND NOT gDevice.stMachineConfig.bPassthrough AND NOT (gDevice.stMachineConfig.tRowCompleteSignalTimeOut = t#0ms), bInhibitReset := FALSE, bInternalReset := FALSE, aAlarmsSettings := gMessage.aAlarmsSettings, nAlarmIndex := nAlarmIndex, sMsgInfo := gMessage.stAlarmTable.aMsgHMI[nAlarmIndex], stMsgAux := gMessage.stAlarmTable.aMsgAux[nAlarmIndex]);

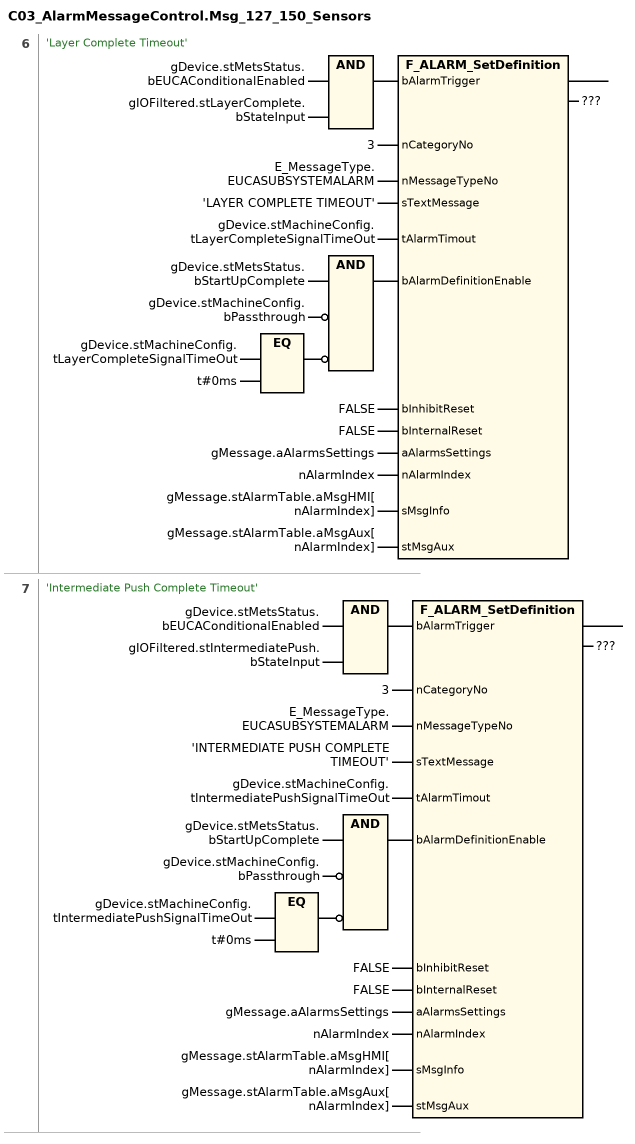
// NETWORK 6
// 'Layer Complete Timeout'
F_ALARM_SetDefinition(bAlarmTrigger := gDevice.stMetsStatus.bEUCAConditionalEnabled AND gIOFiltered.stLayerComplete.bStateInput, nCategoryNo := 3, nMessageTypeNo := E_MessageType.EUCASUBSYSTEMALARM, sTextMessage := 'LAYER COMPLETE TIMEOUT', tAlarmTimout := gDevice.stMachineConfig.tLayerCompleteSignalTimeOut, bAlarmDefinitionEnable := gDevice.stMetsStatus.bStartUpComplete AND NOT gDevice.stMachineConfig.bPassthrough AND NOT (gDevice.stMachineConfig.tLayerCompleteSignalTimeOut = t#0ms), bInhibitReset := FALSE, bInternalReset := FALSE, aAlarmsSettings := gMessage.aAlarmsSettings, nAlarmIndex := nAlarmIndex, sMsgInfo := gMessage.stAlarmTable.aMsgHMI[nAlarmIndex], stMsgAux := gMessage.stAlarmTable.aMsgAux[nAlarmIndex]);

// NETWORK 7
// 'Intermediate Push Complete Timeout'
F_ALARM_SetDefinition(bAlarmTrigger := gDevice.stMetsStatus.bEUCAConditionalEnabled AND gIOFiltered.stIntermediatePush.bStateInput, nCategoryNo := 3, nMessageTypeNo := E_MessageType.EUCASUBSYSTEMALARM, sTextMessage := 'INTERMEDIATE PUSH COMPLETE TIMEOUT', tAlarmTimout := gDevice.stMachineConfig.tIntermediatePushSignalTimeOut, bAlarmDefinitionEnable := gDevice.stMetsStatus.bStartUpComplete AND NOT gDevice.stMachineConfig.bPassthrough AND NOT (gDevice.stMachineConfig.tIntermediatePushSignalTimeOut = t#0ms), bInhibitReset := FALSE, bInternalReset := FALSE, aAlarmsSettings := gMessage.aAlarmsSettings, nAlarmIndex := nAlarmIndex, sMsgInfo := gMessage.stAlarmTable.aMsgHMI[nAlarmIndex], stMsgAux := gMessage.stAlarmTable.aMsgAux[nAlarmIndex]);

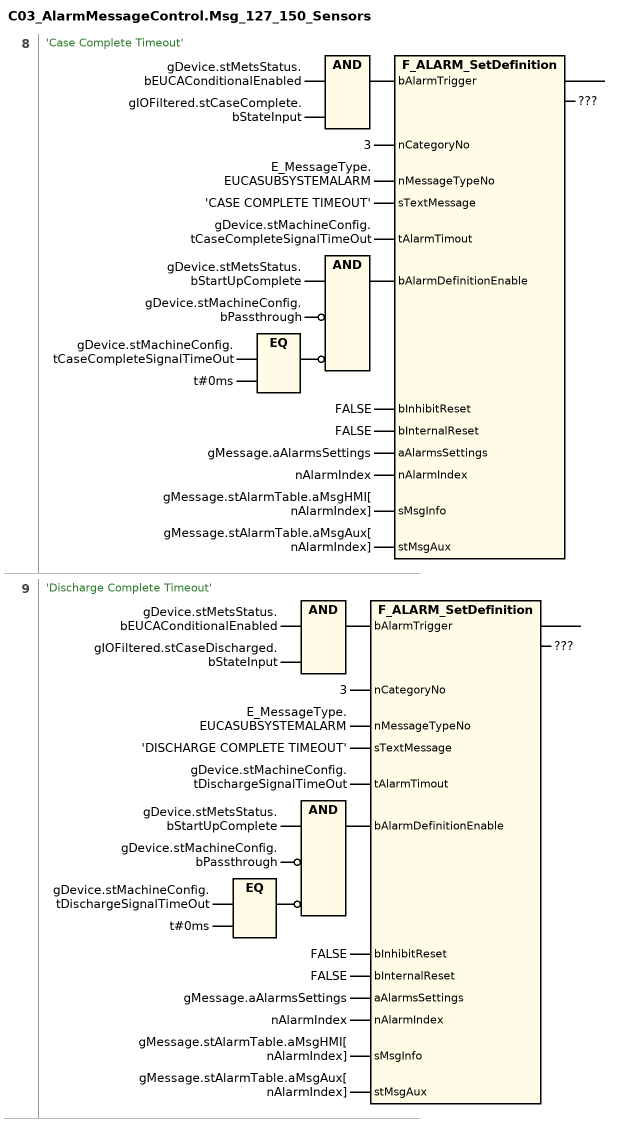
// NETWORK 8
// 'Case Complete Timeout'
F_ALARM_SetDefinition(bAlarmTrigger := gDevice.stMetsStatus.bEUCAConditionalEnabled AND gIOFiltered.stCaseComplete.bStateInput, nCategoryNo := 3, nMessageTypeNo := E_MessageType.EUCASUBSYSTEMALARM, sTextMessage := 'CASE COMPLETE TIMEOUT', tAlarmTimout := gDevice.stMachineConfig.tCaseCompleteSignalTimeOut, bAlarmDefinitionEnable := gDevice.stMetsStatus.bStartUpComplete AND NOT gDevice.stMachineConfig.bPassthrough AND NOT (gDevice.stMachineConfig.tCaseCompleteSignalTimeOut = t#0ms), bInhibitReset := FALSE, bInternalReset := FALSE, aAlarmsSettings := gMessage.aAlarmsSettings, nAlarmIndex := nAlarmIndex, sMsgInfo := gMessage.stAlarmTable.aMsgHMI[nAlarmIndex], stMsgAux := gMessage.stAlarmTable.aMsgAux[nAlarmIndex]);

// NETWORK 9
// 'Discharge Complete Timeout'
F_ALARM_SetDefinition(bAlarmTrigger := gDevice.stMetsStatus.bEUCAConditionalEnabled AND gIOFiltered.stCaseDischarged.bStateInput, nCategoryNo := 3, nMessageTypeNo := E_MessageType.EUCASUBSYSTEMALARM, sTextMessage := 'DISCHARGE COMPLETE TIMEOUT', tAlarmTimout := gDevice.stMachineConfig.tDischargeSignalTimeOut, bAlarmDefinitionEnable := gDevice.stMetsStatus.bStartUpComplete AND NOT gDevice.stMachineConfig.bPassthrough AND NOT (gDevice.stMachineConfig.tDischargeSignalTimeOut = t#0ms), bInhibitReset := FALSE, bInternalReset := FALSE, aAlarmsSettings := gMessage.aAlarmsSettings, nAlarmIndex := nAlarmIndex, sMsgInfo := gMessage.stAlarmTable.aMsgHMI[nAlarmIndex], stMsgAux := gMessage.stAlarmTable.aMsgAux[nAlarmIndex]);

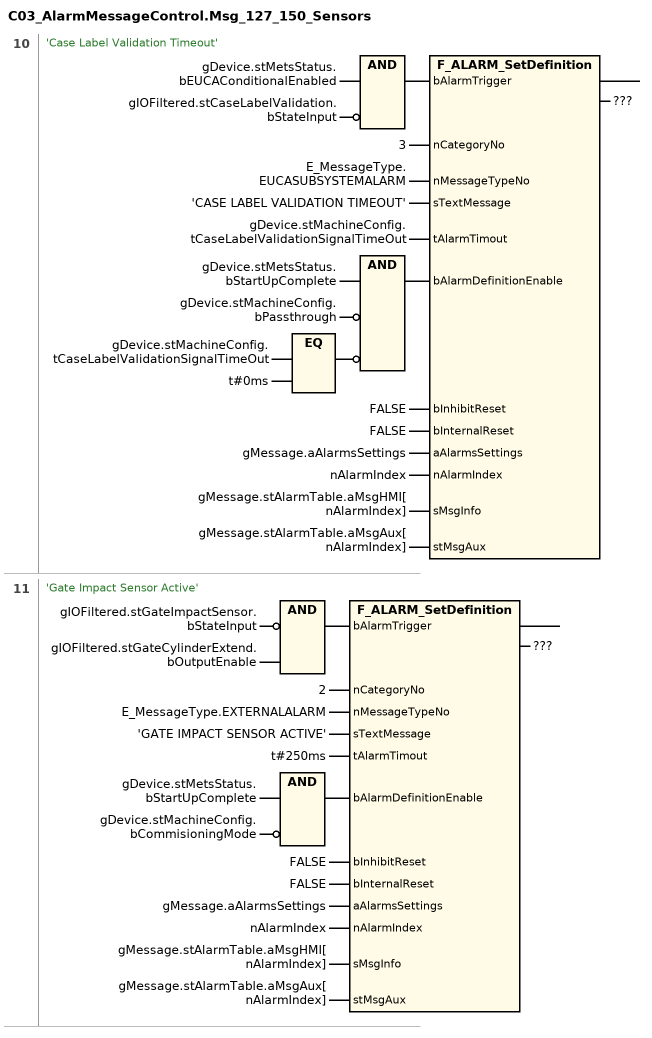
// NETWORK 10
// 'Case Label Validation Timeout'
F_ALARM_SetDefinition(bAlarmTrigger := gDevice.stMetsStatus.bEUCAConditionalEnabled AND NOT gIOFiltered.stCaseLabelValidation.bStateInput, nCategoryNo := 3, nMessageTypeNo := E_MessageType.EUCASUBSYSTEMALARM, sTextMessage := 'CASE LABEL VALIDATION TIMEOUT', tAlarmTimout := gDevice.stMachineConfig.tCaseLabelValidationSignalTimeOut, bAlarmDefinitionEnable := gDevice.stMetsStatus.bStartUpComplete AND NOT gDevice.stMachineConfig.bPassthrough AND NOT (gDevice.stMachineConfig.tCaseLabelValidationSignalTimeOut = t#0ms), bInhibitReset := FALSE, bInternalReset := FALSE, aAlarmsSettings := gMessage.aAlarmsSettings, nAlarmIndex := nAlarmIndex, sMsgInfo := gMessage.stAlarmTable.aMsgHMI[nAlarmIndex], stMsgAux := gMessage.stAlarmTable.aMsgAux[nAlarmIndex]);

// NETWORK 11
// 'Gate Impact Sensor Active'
F_ALARM_SetDefinition(bAlarmTrigger := NOT gIOFiltered.stGateImpactSensor.bStateInput AND gIOFiltered.stGateCylinderExtend.bOutputEnable, nCategoryNo := 2, nMessageTypeNo := E_MessageType.EXTERNALALARM, sTextMessage := 'GATE IMPACT SENSOR ACTIVE', tAlarmTimout := t#250ms, bAlarmDefinitionEnable := gDevice.stMetsStatus.bStartUpComplete AND NOT gDevice.stMachineConfig.bCommisioningMode, bInhibitReset := FALSE, bInternalReset := FALSE, aAlarmsSettings := gMessage.aAlarmsSettings, nAlarmIndex := nAlarmIndex, sMsgInfo := gMessage.stAlarmTable.aMsgHMI[nAlarmIndex], stMsgAux := gMessage.stAlarmTable.aMsgAux[nAlarmIndex]);

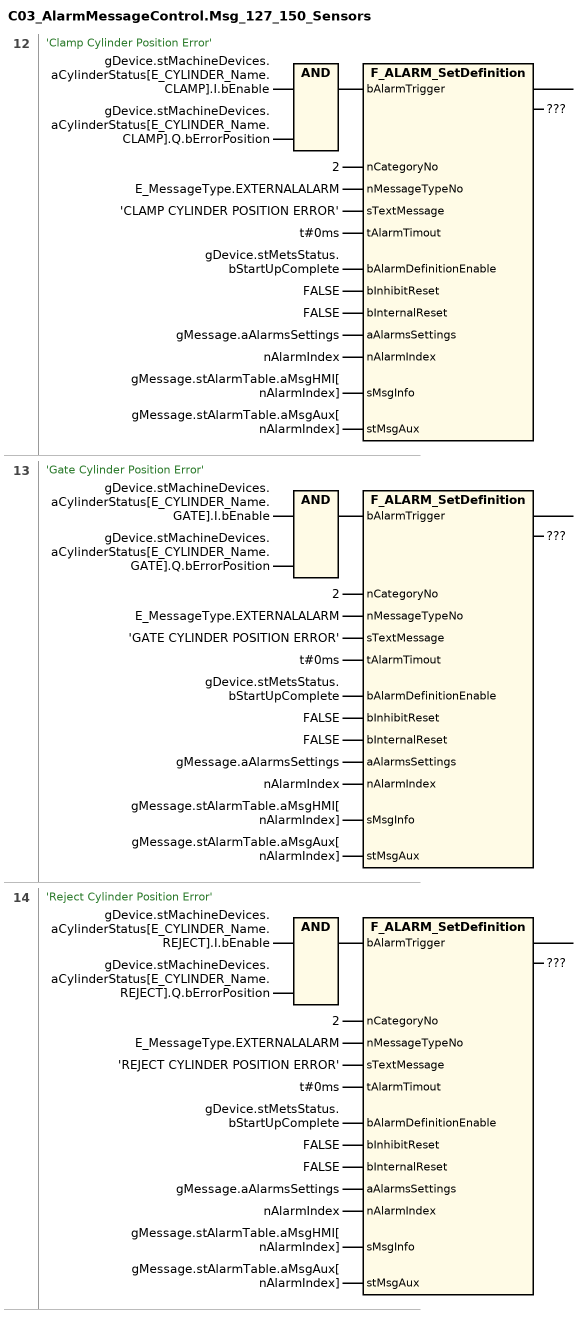
// NETWORK 12
// 'Clamp Cylinder Position Error'
F_ALARM_SetDefinition(bAlarmTrigger := gDevice.stMachineDevices.aCylinderStatus[E_CYLINDER_Name.CLAMP].I.bEnable AND gDevice.stMachineDevices.aCylinderStatus[E_CYLINDER_Name.CLAMP].Q.bErrorPosition, nCategoryNo := 2, nMessageTypeNo := E_MessageType.EXTERNALALARM, sTextMessage := 'CLAMP CYLINDER POSITION ERROR', tAlarmTimout := t#0ms, bAlarmDefinitionEnable := gDevice.stMetsStatus.bStartUpComplete, bInhibitReset := FALSE, bInternalReset := FALSE, aAlarmsSettings := gMessage.aAlarmsSettings, nAlarmIndex := nAlarmIndex, sMsgInfo := gMessage.stAlarmTable.aMsgHMI[nAlarmIndex], stMsgAux := gMessage.stAlarmTable.aMsgAux[nAlarmIndex]);

// NETWORK 13
// 'Gate Cylinder Position Error'
F_ALARM_SetDefinition(bAlarmTrigger := gDevice.stMachineDevices.aCylinderStatus[E_CYLINDER_Name.GATE].I.bEnable AND gDevice.stMachineDevices.aCylinderStatus[E_CYLINDER_Name.GATE].Q.bErrorPosition, nCategoryNo := 2, nMessageTypeNo := E_MessageType.EXTERNALALARM, sTextMessage := 'GATE CYLINDER POSITION ERROR', tAlarmTimout := t#0ms, bAlarmDefinitionEnable := gDevice.stMetsStatus.bStartUpComplete, bInhibitReset := FALSE, bInternalReset := FALSE, aAlarmsSettings := gMessage.aAlarmsSettings, nAlarmIndex := nAlarmIndex, sMsgInfo := gMessage.stAlarmTable.aMsgHMI[nAlarmIndex], stMsgAux := gMessage.stAlarmTable.aMsgAux[nAlarmIndex]);

// NETWORK 14
// 'Reject Cylinder Position Error'
F_ALARM_SetDefinition(bAlarmTrigger := gDevice.stMachineDevices.aCylinderStatus[E_CYLINDER_Name.REJECT].I.bEnable AND gDevice.stMachineDevices.aCylinderStatus[E_CYLINDER_Name.REJECT].Q.bErrorPosition, nCategoryNo := 2, nMessageTypeNo := E_MessageType.EXTERNALALARM, sTextMessage := 'REJECT CYLINDER POSITION ERROR', tAlarmTimout := t#0ms, bAlarmDefinitionEnable := gDevice.stMetsStatus.bStartUpComplete, bInhibitReset := FALSE, bInternalReset := FALSE, aAlarmsSettings := gMessage.aAlarmsSettings, nAlarmIndex := nAlarmIndex, sMsgInfo := gMessage.stAlarmTable.aMsgHMI[nAlarmIndex], stMsgAux := gMessage.stAlarmTable.aMsgAux[nAlarmIndex]);

